// TIA Portal V19 export
DATA_BLOCK "MwFacCalc_GripperEnc"   // DB39
// stored: InstanceOfName ExternalEncoder, InstanceOfType FB
"ExternalEncoder"
   // VAR_INPUT
   //    EncoderCtrl : "TExtEncoder_Ctrl";
   // END_VAR
   // VAR_OUTPUT
   //    EncoderSts : "TExtEncoder_Sts";
   // END_VAR
   // VAR_IN_OUT
   //    TO_Encoder : TO_ExternalEncoder;
   //    Alarm : "TExtEncoder_Alarms";
   //    Diag : "TO_Diagnostic";
   // END_VAR
   // VAR
   //    Status : UInt;
   //    PrevPos : LReal;
   //    POWER : MC_POWER;
   //    RESET : MC_RESET;
   //    HOME : MC_HOME;
   //    TO_Status : "TExtEncoder_StatusWord";
   //    TO_Errors : "TExtEncoder_ErrorWord";
   //    tonTimeOut : IEC_TIMER;
   //    tonStandstill : IEC_TIMER;
   //    Sts : Struct
   //       AlarmPresence : Bool;
   //       Standstill : Bool;
   //       MC_Power_IDLE : Bool;
   //       MC_Reset_IDLE : Bool;
   //       MC_Home_IDLE : Bool;
   //    END_STRUCT;
   //    Local : Struct
   //       RestartConditions : Bool;
   //       ErrorMC_Reset : Bool;
   //       ErrorMC_Power : Bool;
   //       ErrorMC_Home : Bool;
   //    END_STRUCT;
   // END_VAR
BEGIN
END_DATA_BLOCK
